(*
    This function block holds all data that defines a test.
*)
FUNCTION_BLOCK FB_Test
VAR
    TestName : Tc2_System.T_MaxString;
    TestHasFailed : BOOL; // Indication of whether this test has had at least one failed assert
END_VAR

METHOD PUBLIC GetName : Tc2_System.T_MaxString;
GetName := TestName;
END_METHOD

METHOD PUBLIC IsFailed : BOOL
IsFailed := TestHasFailed;
END_METHOD

METHOD PUBLIC SetFailed
TestHasFailed := TRUE;
END_METHOD

METHOD PUBLIC SetName
VAR_INPUT
    Name : Tc2_System.T_MaxString;
END_VAR
TestName := Name;
END_METHOD

END_FUNCTION_BLOCK

(* stored: Version 1.1.0.1, ProductVersion 3.1.4022.12
   POU FB_Test: Id {a51e9086-33ec-4162-acad-93a76961e893}, SpecialFunc None
   Method GetName: Id {94757f0e-9979-49d0-ad9f-e35c823175d4}
   Method IsFailed: Id {e42409e3-251f-4133-8b14-3630785983d6}
   Method SetFailed: Id {b840b41b-4045-4fd9-b97d-0bf226c46fb3}
   Method SetName: Id {4c12f6eb-bbe4-4872-ac89-4411e2e81414} *)
